FUNCTION_BLOCK TEST_SUB2 (* Test SUB functions *)
  (* Standard: IEC 61499-1 *)
  (* Version 0.0, 2006-09-11, JHC, Holobloc Inc *)
  (* Compiler header: package fb.rt.test; *)
  (* Compiler classdef: SimpleFB *)
  (* Compiler Java Sun JDK 1.5.0 *)
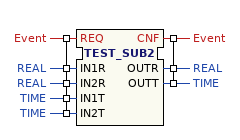
  EVENT_INPUT
    REQ WITH IN1R, IN2R, IN2T, IN1T;
  END_EVENT
  EVENT_OUTPUT
    CNF WITH OUTR, OUTT;
  END_EVENT
  VAR_INPUT
    IN1R : REAL;
    IN2R : REAL;
    IN1T : TIME;
    IN2T : TIME;
  END_VAR
  VAR_OUTPUT
    OUTR : REAL;
    OUTT : TIME;
  END_VAR
  ALGORITHM REQ IN FBD:
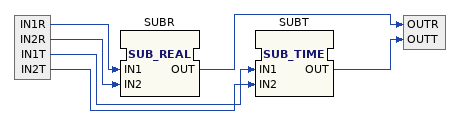
    FBS
      SUBR : SUB_REAL;
      SUBT : SUB_TIME;
    END_FBS
    DATA_CONNECTIONS
      IN1R TO SUBR.IN1;
      IN2R TO SUBR.IN2;
      SUBR.OUT TO OUTR;
      IN1T TO SUBT.IN1;
      IN2T TO SUBT.IN2;
      SUBT.OUT TO OUTT;
    END_CONNECTIONS
  END_ALGORITHM
END_FUNCTION_BLOCK
